FUNCTION_BLOCK Softkey_IE (* Input service interface function block for event input data *)
  (* Description: Copyright (c) 2014, 2023 fortiss GmbH, HR Agrartechnik GmbH This program and the accompanying materials are made available under the terms of the Eclipse Public License 2.0 which is available at https://www.eclipse.org/legal/epl-2.0/ SPDX-License-Identifier: EPL-2.0 *)
  (* Version 1.0, 2014-08-26, Waldemar Eisenmenger, fortiss GmbH *)
  (* Version 1.1, 2014-08-30, Alois Zoitl, fortiss GmbH *)
  (* Version 1.2, 2015-06-10, Monika Wenger, fortiss GmbH *)
  (* Version 1.3, 2023-09-07, Franz Höpfinger, HR Agrartechnik GmbH *)
  PACKAGE isobus::UT::io::Softkey;
  IMPORT eclipse4diac::core::TypeHash;
  IMPORT isobus::UT::Q::const::IDs::ID_NULL;
  IMPORT isobus::UT::io::Softkey::SoftKeyActivationCode::Invalid;
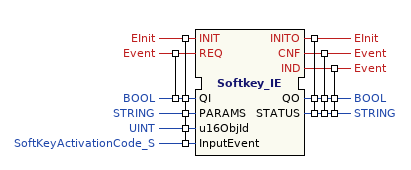
  EVENT_INPUT
    INIT : EInit WITH QI, PARAMS, u16ObjId, InputEvent; (* Service Initialization *)
    REQ WITH QI; (* Service Request *)
  END_EVENT
  EVENT_OUTPUT
    INITO : EInit WITH QO, STATUS; (* Initialization Confirm *)
    CNF WITH QO, STATUS; (* Confirmation of Requested Service *)
    IND WITH QO, STATUS; (* Indication from Resource *)
  END_EVENT
  VAR_INPUT
    QI : BOOL; (* Event Input Qualifier *)
    PARAMS : STRING; (* Service Parameters *)
    u16ObjId : UINT := ID_NULL; (* Object ID *)
    InputEvent : isobus::UT::io::Softkey::SoftKeyActivationCode_S := Invalid; (* Identify the Event according to ISO 11783-6 *)
  END_VAR
  VAR_OUTPUT
    QO : BOOL; (* Event Output Qualifier *)
    STATUS : STRING; (* Service Status *)
  END_VAR
END_FUNCTION_BLOCK
